// TIA Portal project "Project" (V13)

(* hardware
DEVICE "S7300/ET200M station_1"  S7-300 station
   slot 0: "Rail_0"  Rail  6ES7 390-1***0-0AA0
   slot 1: "PS 307 2A_1"  PS 307 2A  6ES7 307-1BA00-0AA0
   slot 2: "PLC-241"  CPU 315-2 PN/DP  6ES7 315-2EH13-0AB0  V2.6
      slot 1: "MPI/DP interface_1"  X1
      slot 2: "PROFINET interface_1"  PN-IO
         slot 1: "Port_1"  Port
   slot 4: "DI 16/DO 16x24VDC/0.5A_1"  DI16/DO16 x 24V / 0.5A  6ES7 323-1BL00-0AA0
DEVICE "PC-System_1"  SIMATIC PC station
   slot 0: "SIMATIC PC station"  Rail  SIMATIC PC-Station  V1.0
      slot 125: "Stationmanager"  Station_Manager  V6.0.4
   slot 1: "HMI_RT_1"  WinCC RT Advanced  6AV2 104-0xxxx-xxxx  13.0.1.0
      slot 33792: "Host interface"  Host interface
   slot 2: "IE general_1"  IE General  IE_CP  V8.2.0
*)

// ===== PLC "PLC-241"  CPU 315-2 PN/DP =====

VAR_GLOBAL   // PLC tag table "Default tag table"
   "tipka_crna_L_zgoraj" AT %I1.4 : Bool;
   "tipka_crna_L_spodaj" AT %I1.5 : Bool;
   "tipka_crna_D_zgoraj" AT %I1.6 : Bool;
   "tipka_crna_D_spodaj" AT %I1.7 : Bool;
   "kljuc" AT %I1.2 : Bool;
   "tipka_zelena" AT %I1.3 : Bool;
   "vrtljivaMiza_R_vhod" AT %I0.0 : Bool;
   "vrtljivaMiza_I_vhod" AT %I0.1 : Bool;
   "teleskopskaRoka_R_vhod" AT %I0.2 : Bool;
   "teleskopskaRoka_I_vhod" AT %I0.3 : Bool;
   "dvig_R_vhod" AT %I0.4 : Bool;
   "dvig_I_vhod" AT %I0.5 : Bool;
   "prijemalo_R_vhod" AT %I0.6 : Bool;
   "prijemalo_I_vhod" AT %I0.7 : Bool;
   "vrtljivaMiza_S_izhod" AT %Q0.0 : Bool;
   "vrtljivaMiza_P_izhod" AT %Q0.1 : Bool;
   "teleskopskaRoka_S_izhod" AT %Q0.2 : Bool;
   "teleskopskaRoka_P_izhod" AT %Q0.3 : Bool;
   "dvig_S_izhod" AT %Q0.4 : Bool;
   "dvig_P_izhod" AT %Q0.5 : Bool;
   "prijemalo_S_izhod" AT %Q0.6 : Bool;
   "prijemalo_P_izhod" AT %Q0.7 : Bool;
   "lucka_rdeca_L" AT %Q1.4 : Bool;
   "lucka_rumena_L" AT %Q1.5 : Bool;
   "lucka_rdeca_D" AT %Q1.6 : Bool;
   "lucka_rumena_D" AT %Q1.7 : Bool;
   "s" AT %M2.0 : Bool;
   "memory_1" AT %M4.0 : Bool;
   "memory_2" AT %M6.0 : Bool;
END_VAR

TYPE "Lokacija"
   STRUCT
      "ID izdelka" : Int;
      koordinate : "Koordinate";
   END_STRUCT;
END_TYPE

TYPE "Koordinate"
   STRUCT
      miza : Int;
      izteg : Int;
      dvig : Int;
      stisk : Int;
   END_STRUCT;
END_TYPE

DATA_BLOCK "spremenljivke"   // DB1
{ S7_Optimized_Access := 'FALSE' }
VERSION : 0.1
   VAR
      smer : Bool;
      premik : Bool;
      auto_motor1_ccw : Bool;
      auto_motor1_cw : Bool;
      izbiraMotorja : Int;
      levo : Bool;
      desno : Bool;
      vrtljivaMiza_TRENUTNO : Int;
      teleskopskaRoka_TRENUTNO : Int;
      dvig_TRENUTNO : Int;
      premik_TRENUTNO : Int;
      dvig_max : Int;
      vrtljivaMiza_max : Int;
      premik_max : Int;
      teleskopskaRoka_MAX : Int;
      Recept_prej : Int;
      stevecLokacij : Int;
      neki : Int;
      izdelekID : Int;
      izbiraRecepta : Int;
      stevecKosov : Int;
      prva_ref_roka : Bool;
      prva_ref_dvig : Bool;
      prva_ref_stisk : Bool;
      prva_ref_miza : Bool;
      prva_rs_dvig : Bool;
      prva_rs_stisk : Bool;
      prva_rs_roka : Bool;
      prva_rs_miza : Bool;
      miza_ok : Bool;
      stisk_ok : Bool;
      roka_ok : Bool;
      dvig_ok : Bool;
      razlika_dvig : Int;
      razlika_miza : Int;
      razlika_stisk : Int;
      razlika_roka : Int;
   END_VAR
BEGIN
END_DATA_BLOCK

DATA_BLOCK "Motor_DB_1"   // DB2
{ S7_Optimized_Access := 'FALSE' }
VERSION : 0.1
// stored: InstanceOfName Motor
"Motor"
BEGIN
END_DATA_BLOCK

DATA_BLOCK "Lokacije"   // DB3
{ S7_Optimized_Access := 'FALSE' }
VERSION : 0.1
   VAR
      lokacija0 : "Lokacija";
      lokacija1 : "Lokacija";
      lokacija2 : "Lokacija";
      lokacija3 : "Lokacija";
      lokacija4 : "Lokacija";
      lokacija5 : "Lokacija";
      lokacija6 : "Lokacija";
      lokacija7 : "Lokacija";
   END_VAR
BEGIN
END_DATA_BLOCK

DATA_BLOCK "vrtljivaMiza_DB"   // DB4
{ S7_Optimized_Access := 'FALSE' }
VERSION : 0.1
// stored: InstanceOfName vrtljivaMiza
"vrtljivaMiza"
BEGIN
END_DATA_BLOCK

DATA_BLOCK "stevecMotorjev_DB_1"   // DB5
{ S7_Optimized_Access := 'FALSE' }
VERSION : 0.1
// stored: InstanceOfName stevecMotorjev
"stevecMotorjev"
BEGIN
END_DATA_BLOCK

DATA_BLOCK "teleskopskaRoka_DB"   // DB6
{ S7_Optimized_Access := 'FALSE' }
VERSION : 0.1
// stored: InstanceOfName teleskopskaRoka
"teleskopskaRoka"
BEGIN
END_DATA_BLOCK

DATA_BLOCK "dvig_DB"   // DB7
{ S7_Optimized_Access := 'FALSE' }
VERSION : 0.1
// stored: InstanceOfName dvig
"dvig"
BEGIN
END_DATA_BLOCK

DATA_BLOCK "prijemalo_DB"   // DB8
{ S7_Optimized_Access := 'FALSE' }
VERSION : 0.1
// stored: InstanceOfName prijemalo
"prijemalo"
BEGIN
END_DATA_BLOCK

DATA_BLOCK "TrenutnaLokacija"   // DB9
{ S7_Optimized_Access := 'FALSE' }
VERSION : 0.1
   VAR
      lokacija : "Lokacija";
   END_VAR
BEGIN
END_DATA_BLOCK

DATA_BLOCK "IzbiraLokacije_DB"   // DB10
{ S7_Optimized_Access := 'FALSE' }
VERSION : 0.1
// stored: InstanceOfName IzbiraLokacije
"IzbiraLokacije"
BEGIN
END_DATA_BLOCK

DATA_BLOCK "IzbiraLokacije_DB_1"   // DB11
{ S7_Optimized_Access := 'FALSE' }
VERSION : 0.1
// stored: InstanceOfName IzbiraLokacije
"IzbiraLokacije"
BEGIN
END_DATA_BLOCK

DATA_BLOCK "Recept 1"   // DB12
{ S7_Optimized_Access := 'FALSE' }
VERSION : 0.1
   VAR
      lokacija10 : "Lokacija";
      lokacija11 : "Lokacija";
      lokacija12 : "Lokacija";
      lokacija13 : "Lokacija";
      lokacija14 : "Lokacija";
      lokacija15 : "Lokacija";
      lokacija16 : "Lokacija";
      lokacija17 : "Lokacija";
   END_VAR
BEGIN
END_DATA_BLOCK

DATA_BLOCK "Recept 2"   // DB13
{ S7_Optimized_Access := 'FALSE' }
VERSION : 0.1
   VAR
      lokacija20 : "Lokacija";
      lokacija21 : "Lokacija";
      lokacija22 : "Lokacija";
      lokacija23 : "Lokacija";
      lokacija24 : "Lokacija";
      lokacija25 : "Lokacija";
      lokacija26 : "Lokacija";
      lokacija27 : "Lokacija";
   END_VAR
BEGIN
END_DATA_BLOCK

DATA_BLOCK "Alarmi"   // DB14
{ S7_Optimized_Access := 'FALSE' }
VERSION : 0.1
   VAR
      alarmi : Array[0..15] of Bool;
      alarmPotrdi : Bool;
      alarmRS1 : Bool;
      alarmRS2 : Bool;
      alarmRS3 : Bool;
      alarmRS4 : Bool;
      alarmRS5 : Bool;
      alarmRS6 : Bool;
      Globalni_alarm : Bool;
   END_VAR
BEGIN
END_DATA_BLOCK

DATA_BLOCK "izbiraAlarmov_DB"   // DB15
{ S7_Optimized_Access := 'FALSE' }
VERSION : 0.1
// stored: InstanceOfName izbiraAlarmov
"izbiraAlarmov"
BEGIN
END_DATA_BLOCK

FUNCTION_BLOCK "Motor"   // FB1, LAD
{ S7_Optimized_Access := 'FALSE' }
VERSION : 0.1
   VAR_TEMP   // added for the SCL form of the ladder/FBD networks
      _w1 : Bool;
      _w2 : Bool;
   END_VAR
BEGIN

REGION Network 1
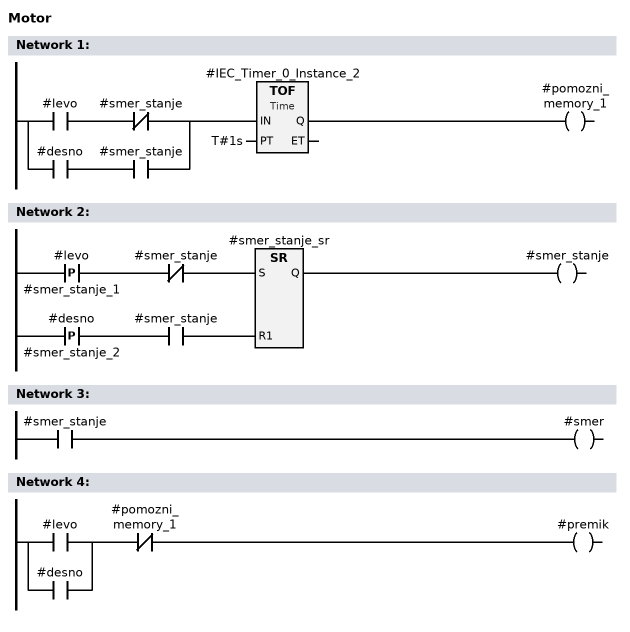
   #IEC_Timer_0_Instance_2.TOF(IN := (#levo AND NOT #smer_stanje) OR (#desno AND #smer_stanje), PT := T#1s);
   #pomozni_memory_1 := #IEC_Timer_0_Instance_2.Q;
END_REGION

REGION Network 2
   RUNG wire#powerrail
      P_Contact(operand := #levo, bit := #smer_stanje_1)
      I_Contact( #smer_stanje )
      S_SR(operand := #smer_stanje_sr, r1 := wire#w1)
      Coil( #smer_stanje )
   END_RUNG
   RUNG wire#powerrail
      P_Contact(operand := #desno, bit := #smer_stanje_2)
      Contact( #smer_stanje )
   END_RUNG wire#w1
   // the same network as SCL:
   #_w1 := #levo AND NOT #smer_stanje_1;   // rising edge of #levo
   #smer_stanje_1 := #levo;
   #_w2 := #desno AND NOT #smer_stanje_2;   // rising edge of #desno
   #smer_stanje_2 := #desno;
   IF #_w1 AND NOT #smer_stanje THEN
       #smer_stanje_sr := TRUE;   // SR flip-flop
   END_IF;
   IF #_w2 AND #smer_stanje THEN #smer_stanje_sr := FALSE; END_IF;
   #smer_stanje := #smer_stanje_sr;
END_REGION

REGION Network 3
   RUNG wire#powerrail
      Contact( #smer_stanje )
      Coil( #smer )
   END_RUNG
   // the same network as SCL:
   #smer := #smer_stanje;
END_REGION

REGION Network 4
   RUNG wire#powerrail
      Contact( #levo )
      wire#w1
      I_Contact( #pomozni_memory_1 )
      Coil( #premik )
   END_RUNG
   RUNG wire#powerrail
      Contact( #desno )
   END_RUNG wire#w1
   // the same network as SCL:
   #premik := (#levo OR #desno) AND NOT #pomozni_memory_1;
END_REGION
END_FUNCTION_BLOCK

FUNCTION_BLOCK "stevecMotorjev"   // FB2, LAD
{ S7_Optimized_Access := 'FALSE' }
VERSION : 0.1
BEGIN

REGION Network 1
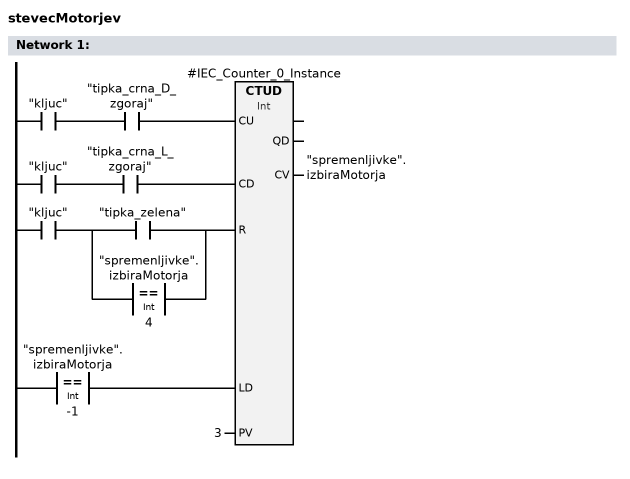
   #IEC_Counter_0_Instance.CTUD(CU := "kljuc" AND "tipka_crna_D_zgoraj",
                           CD := "kljuc" AND "tipka_crna_L_zgoraj",
                           R := "kljuc" AND ("tipka_zelena" OR ("spremenljivke".izbiraMotorja = 4)),
                           LD := "spremenljivke".izbiraMotorja = (-1),
                           PV := 3,
                           CV => "spremenljivke".izbiraMotorja);
END_REGION
END_FUNCTION_BLOCK

FUNCTION_BLOCK "vrtljivaMiza"   // FB3, LAD
{ S7_Optimized_Access := 'FALSE' }
VERSION : 0.1
BEGIN

REGION Network 1
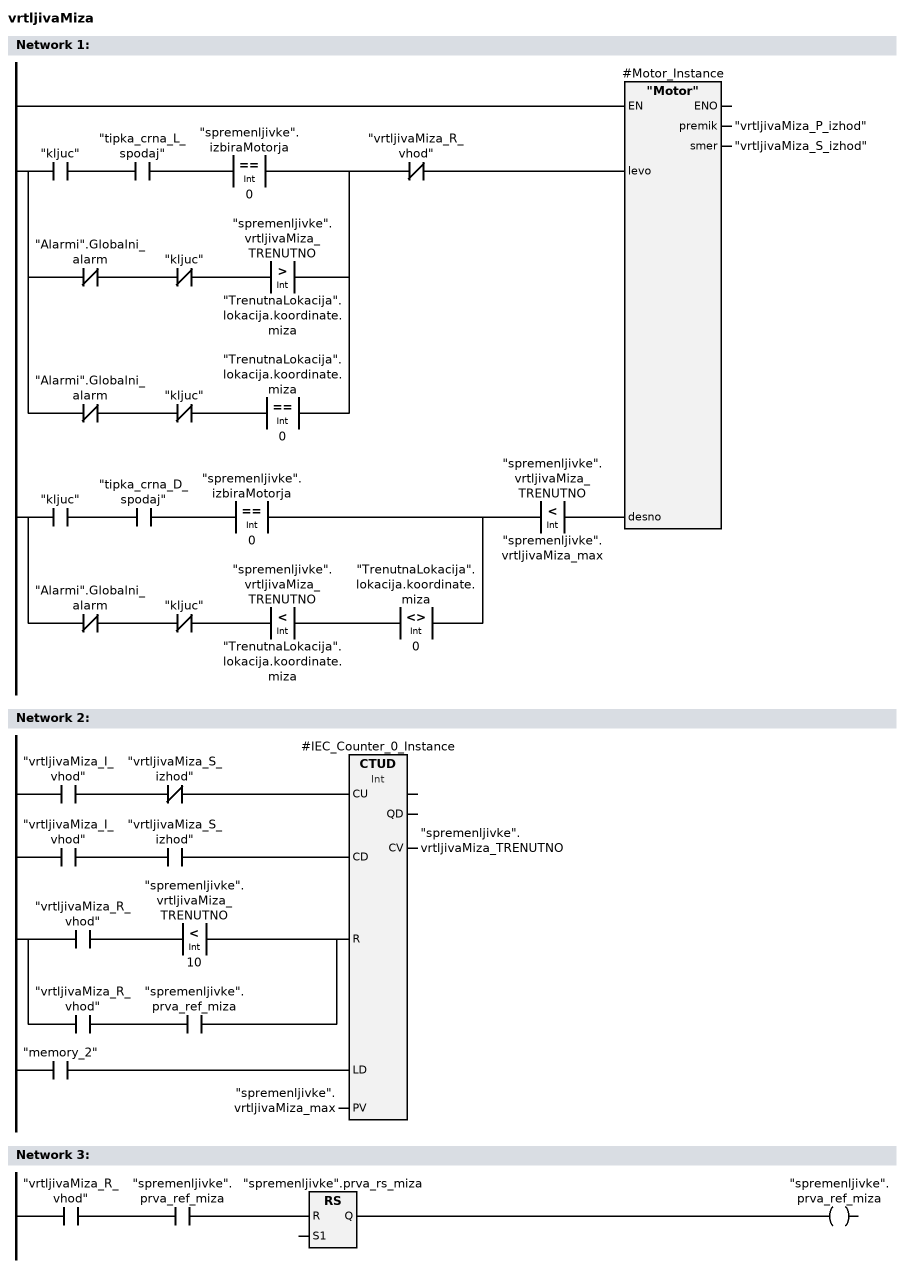
   RUNG wire#powerrail
      #Motor_Instance(levo := wire#w2, desno := wire#w4, premik => "vrtljivaMiza_P_izhod", smer => "vrtljivaMiza_S_izhod")
   END_RUNG
   RUNG wire#powerrail
      Contact( "kljuc" )
      Contact( "tipka_crna_L_spodaj" )
      { S7_Templates := "SrcType := Int" } EQ_Contact(in1 := "spremenljivke".izbiraMotorja, in2 := 0)
      wire#w1
      I_Contact( "vrtljivaMiza_R_vhod" )
   END_RUNG wire#w2
   RUNG wire#powerrail
      I_Contact( "Alarmi".Globalni_alarm )
      I_Contact( "kljuc" )
      { S7_Templates := "SrcType := Int" } GT_Contact(in1 := "spremenljivke".vrtljivaMiza_TRENUTNO, in2 := "TrenutnaLokacija".lokacija.koordinate.miza)
   END_RUNG wire#w1
   RUNG wire#powerrail
      I_Contact( "Alarmi".Globalni_alarm )
      I_Contact( "kljuc" )
      { S7_Templates := "SrcType := Int" } EQ_Contact(in1 := "TrenutnaLokacija".lokacija.koordinate.miza, in2 := 0)
   END_RUNG wire#w1
   RUNG wire#powerrail
      Contact( "kljuc" )
      Contact( "tipka_crna_D_spodaj" )
      { S7_Templates := "SrcType := Int" } EQ_Contact(in1 := "spremenljivke".izbiraMotorja, in2 := 0)
      wire#w3
      { S7_Templates := "SrcType := Int" } LT_Contact(in1 := "spremenljivke".vrtljivaMiza_TRENUTNO, in2 := "spremenljivke".vrtljivaMiza_max)
   END_RUNG wire#w4
   RUNG wire#powerrail
      I_Contact( "Alarmi".Globalni_alarm )
      I_Contact( "kljuc" )
      { S7_Templates := "SrcType := Int" } LT_Contact(in1 := "spremenljivke".vrtljivaMiza_TRENUTNO, in2 := "TrenutnaLokacija".lokacija.koordinate.miza)
      { S7_Templates := "SrcType := Int" } NE_Contact(in1 := "TrenutnaLokacija".lokacija.koordinate.miza, in2 := 0)
   END_RUNG wire#w3
   // the same network as SCL:
   #Motor_Instance(levo := (("kljuc" AND "tipka_crna_L_spodaj" AND ("spremenljivke".izbiraMotorja = 0)) OR (NOT "Alarmi".Globalni_alarm AND NOT "kljuc" AND ("spremenljivke".vrtljivaMiza_TRENUTNO > "TrenutnaLokacija".lokacija.koordinate.miza)) OR (NOT "Alarmi".Globalni_alarm AND NOT "kljuc" AND ("TrenutnaLokacija".lokacija.koordinate.miza = 0))) AND NOT "vrtljivaMiza_R_vhod",   // "Motor"
                   desno := (("kljuc" AND "tipka_crna_D_spodaj" AND ("spremenljivke".izbiraMotorja = 0)) OR (NOT "Alarmi".Globalni_alarm AND NOT "kljuc" AND ("spremenljivke".vrtljivaMiza_TRENUTNO < "TrenutnaLokacija".lokacija.koordinate.miza) AND ("TrenutnaLokacija".lokacija.koordinate.miza <> 0))) AND ("spremenljivke".vrtljivaMiza_TRENUTNO < "spremenljivke".vrtljivaMiza_max),
                   premik => "vrtljivaMiza_P_izhod",
                   smer => "vrtljivaMiza_S_izhod");
END_REGION

REGION Network 2
   #IEC_Counter_0_Instance.CTUD(CU := "vrtljivaMiza_I_vhod" AND NOT "vrtljivaMiza_S_izhod",
                           CD := "vrtljivaMiza_I_vhod" AND "vrtljivaMiza_S_izhod",
                           R := ("vrtljivaMiza_R_vhod" AND ("spremenljivke".vrtljivaMiza_TRENUTNO < 10)) OR ("vrtljivaMiza_R_vhod" AND "spremenljivke".prva_ref_miza),
                           LD := "memory_2",
                           PV := "spremenljivke".vrtljivaMiza_max,
                           CV => "spremenljivke".vrtljivaMiza_TRENUTNO);
END_REGION

REGION Network 3
   RUNG wire#powerrail
      Contact( "vrtljivaMiza_R_vhod" )
      Contact( "spremenljivke".prva_ref_miza )
      S_RS(operand := "spremenljivke".prva_rs_miza, s1 :=)
      Coil( "spremenljivke".prva_ref_miza )
   END_RUNG
   // the same network as SCL:
   IF "vrtljivaMiza_R_vhod" AND "spremenljivke".prva_ref_miza THEN
       "spremenljivke".prva_rs_miza := FALSE;   // RS flip-flop
   END_IF;
   "spremenljivke".prva_ref_miza := "spremenljivke".prva_rs_miza;
END_REGION
END_FUNCTION_BLOCK

FUNCTION_BLOCK "teleskopskaRoka"   // FB4, LAD
{ S7_Optimized_Access := 'FALSE' }
VERSION : 0.1
BEGIN

REGION Network 1
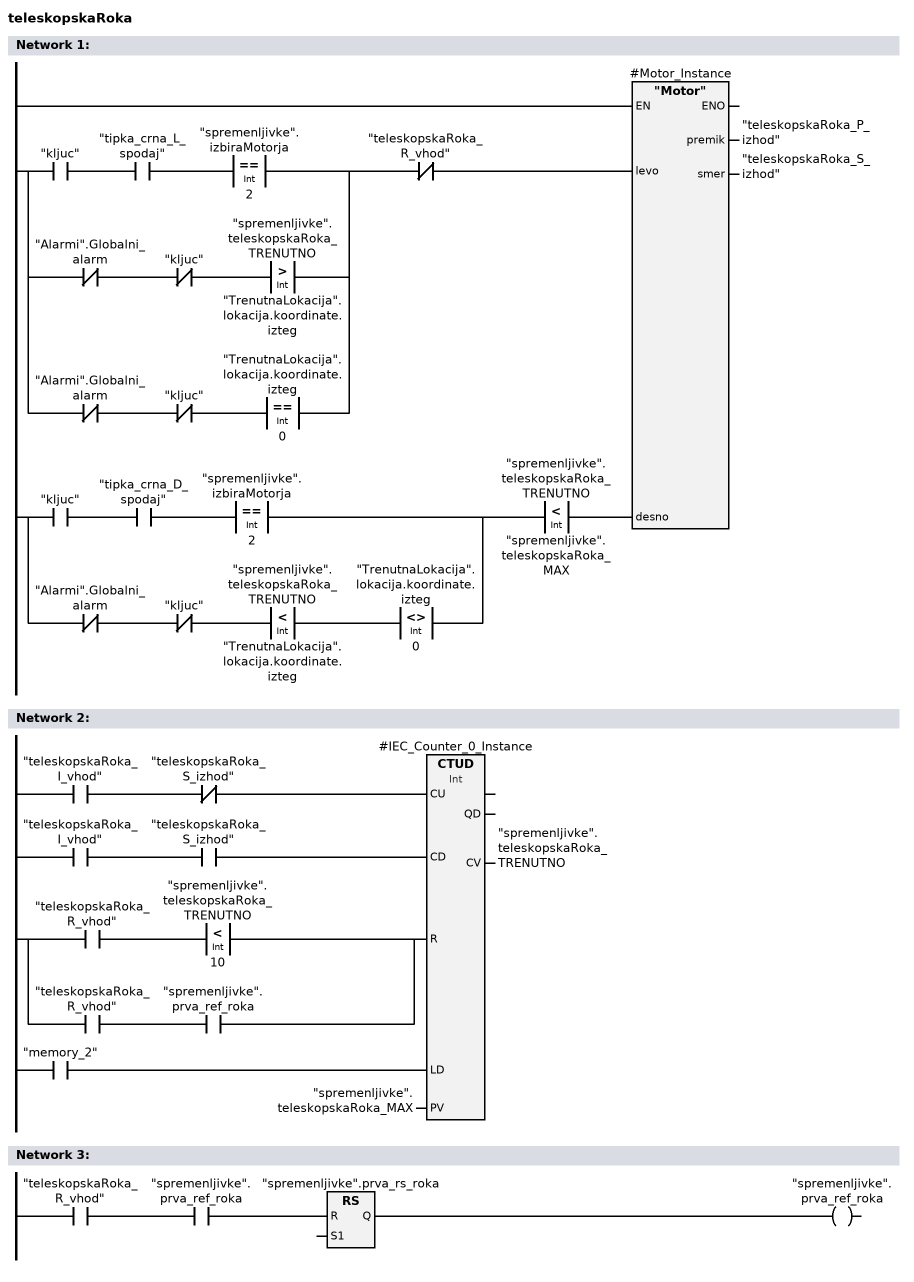
   RUNG wire#powerrail
      #Motor_Instance(levo := wire#w2, desno := wire#w4, premik => "teleskopskaRoka_P_izhod", smer => "teleskopskaRoka_S_izhod")
   END_RUNG
   RUNG wire#powerrail
      Contact( "kljuc" )
      Contact( "tipka_crna_L_spodaj" )
      { S7_Templates := "SrcType := Int" } EQ_Contact(in1 := "spremenljivke".izbiraMotorja, in2 := 2)
      wire#w1
      I_Contact( "teleskopskaRoka_R_vhod" )
   END_RUNG wire#w2
   RUNG wire#powerrail
      I_Contact( "Alarmi".Globalni_alarm )
      I_Contact( "kljuc" )
      { S7_Templates := "SrcType := Int" } GT_Contact(in1 := "spremenljivke".teleskopskaRoka_TRENUTNO, in2 := "TrenutnaLokacija".lokacija.koordinate.izteg)
   END_RUNG wire#w1
   RUNG wire#powerrail
      I_Contact( "Alarmi".Globalni_alarm )
      I_Contact( "kljuc" )
      { S7_Templates := "SrcType := Int" } EQ_Contact(in1 := "TrenutnaLokacija".lokacija.koordinate.izteg, in2 := 0)
   END_RUNG wire#w1
   RUNG wire#powerrail
      Contact( "kljuc" )
      Contact( "tipka_crna_D_spodaj" )
      { S7_Templates := "SrcType := Int" } EQ_Contact(in1 := "spremenljivke".izbiraMotorja, in2 := 2)
      wire#w3
      { S7_Templates := "SrcType := Int" } LT_Contact(in1 := "spremenljivke".teleskopskaRoka_TRENUTNO, in2 := "spremenljivke".teleskopskaRoka_MAX)
   END_RUNG wire#w4
   RUNG wire#powerrail
      I_Contact( "Alarmi".Globalni_alarm )
      I_Contact( "kljuc" )
      { S7_Templates := "SrcType := Int" } LT_Contact(in1 := "spremenljivke".teleskopskaRoka_TRENUTNO, in2 := "TrenutnaLokacija".lokacija.koordinate.izteg)
      { S7_Templates := "SrcType := Int" } NE_Contact(in1 := "TrenutnaLokacija".lokacija.koordinate.izteg, in2 := 0)
   END_RUNG wire#w3
   // the same network as SCL:
   #Motor_Instance(levo := (("kljuc" AND "tipka_crna_L_spodaj" AND ("spremenljivke".izbiraMotorja = 2)) OR (NOT "Alarmi".Globalni_alarm AND NOT "kljuc" AND ("spremenljivke".teleskopskaRoka_TRENUTNO > "TrenutnaLokacija".lokacija.koordinate.izteg)) OR (NOT "Alarmi".Globalni_alarm AND NOT "kljuc" AND ("TrenutnaLokacija".lokacija.koordinate.izteg = 0))) AND NOT "teleskopskaRoka_R_vhod",   // "Motor"
                   desno := (("kljuc" AND "tipka_crna_D_spodaj" AND ("spremenljivke".izbiraMotorja = 2)) OR (NOT "Alarmi".Globalni_alarm AND NOT "kljuc" AND ("spremenljivke".teleskopskaRoka_TRENUTNO < "TrenutnaLokacija".lokacija.koordinate.izteg) AND ("TrenutnaLokacija".lokacija.koordinate.izteg <> 0))) AND ("spremenljivke".teleskopskaRoka_TRENUTNO < "spremenljivke".teleskopskaRoka_MAX),
                   premik => "teleskopskaRoka_P_izhod",
                   smer => "teleskopskaRoka_S_izhod");
END_REGION

REGION Network 2
   #IEC_Counter_0_Instance.CTUD(CU := "teleskopskaRoka_I_vhod" AND NOT "teleskopskaRoka_S_izhod",
                           CD := "teleskopskaRoka_I_vhod" AND "teleskopskaRoka_S_izhod",
                           R := ("teleskopskaRoka_R_vhod" AND ("spremenljivke".teleskopskaRoka_TRENUTNO < 10)) OR ("teleskopskaRoka_R_vhod" AND "spremenljivke".prva_ref_roka),
                           LD := "memory_2",
                           PV := "spremenljivke".teleskopskaRoka_MAX,
                           CV => "spremenljivke".teleskopskaRoka_TRENUTNO);
END_REGION

REGION Network 3
   RUNG wire#powerrail
      Contact( "teleskopskaRoka_R_vhod" )
      Contact( "spremenljivke".prva_ref_roka )
      S_RS(operand := "spremenljivke".prva_rs_roka, s1 :=)
      Coil( "spremenljivke".prva_ref_roka )
   END_RUNG
   // the same network as SCL:
   IF "teleskopskaRoka_R_vhod" AND "spremenljivke".prva_ref_roka THEN
       "spremenljivke".prva_rs_roka := FALSE;   // RS flip-flop
   END_IF;
   "spremenljivke".prva_ref_roka := "spremenljivke".prva_rs_roka;
END_REGION
END_FUNCTION_BLOCK

FUNCTION_BLOCK "dvig"   // FB5, LAD
{ S7_Optimized_Access := 'FALSE' }
VERSION : 0.1
BEGIN

REGION Network 1
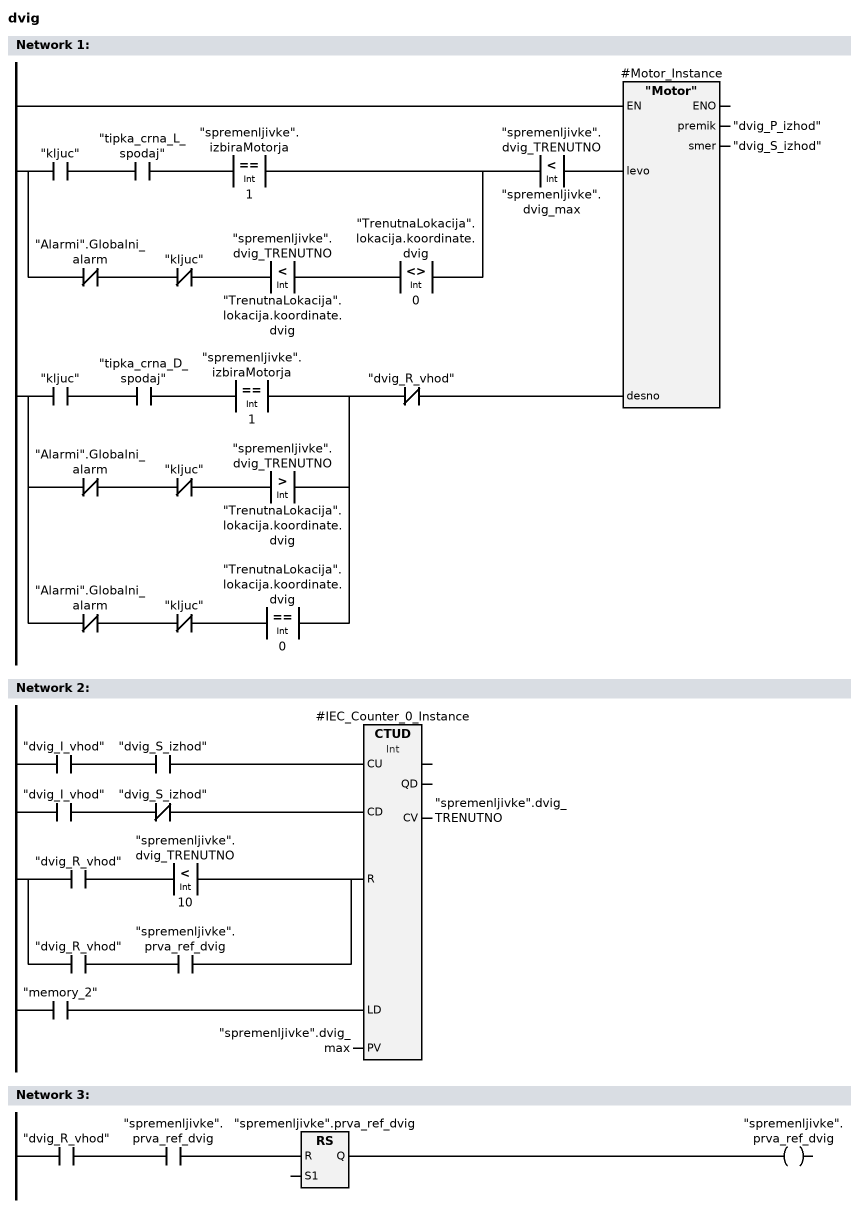
   RUNG wire#powerrail
      #Motor_Instance(levo := wire#w2, desno := wire#w4, premik => "dvig_P_izhod", smer => "dvig_S_izhod")
   END_RUNG
   RUNG wire#powerrail
      Contact( "kljuc" )
      Contact( "tipka_crna_L_spodaj" )
      { S7_Templates := "SrcType := Int" } EQ_Contact(in1 := "spremenljivke".izbiraMotorja, in2 := 1)
      wire#w1
      { S7_Templates := "SrcType := Int" } LT_Contact(in1 := "spremenljivke".dvig_TRENUTNO, in2 := "spremenljivke".dvig_max)
   END_RUNG wire#w2
   RUNG wire#powerrail
      I_Contact( "Alarmi".Globalni_alarm )
      I_Contact( "kljuc" )
      { S7_Templates := "SrcType := Int" } LT_Contact(in1 := "spremenljivke".dvig_TRENUTNO, in2 := "TrenutnaLokacija".lokacija.koordinate.dvig)
      { S7_Templates := "SrcType := Int" } NE_Contact(in1 := "TrenutnaLokacija".lokacija.koordinate.dvig, in2 := 0)
   END_RUNG wire#w1
   RUNG wire#powerrail
      Contact( "kljuc" )
      Contact( "tipka_crna_D_spodaj" )
      { S7_Templates := "SrcType := Int" } EQ_Contact(in1 := "spremenljivke".izbiraMotorja, in2 := 1)
      wire#w3
      I_Contact( "dvig_R_vhod" )
   END_RUNG wire#w4
   RUNG wire#powerrail
      I_Contact( "Alarmi".Globalni_alarm )
      I_Contact( "kljuc" )
      { S7_Templates := "SrcType := Int" } GT_Contact(in1 := "spremenljivke".dvig_TRENUTNO, in2 := "TrenutnaLokacija".lokacija.koordinate.dvig)
   END_RUNG wire#w3
   RUNG wire#powerrail
      I_Contact( "Alarmi".Globalni_alarm )
      I_Contact( "kljuc" )
      { S7_Templates := "SrcType := Int" } EQ_Contact(in1 := "TrenutnaLokacija".lokacija.koordinate.dvig, in2 := 0)
   END_RUNG wire#w3
   // the same network as SCL:
   #Motor_Instance(levo := (("kljuc" AND "tipka_crna_L_spodaj" AND ("spremenljivke".izbiraMotorja = 1)) OR (NOT "Alarmi".Globalni_alarm AND NOT "kljuc" AND ("spremenljivke".dvig_TRENUTNO < "TrenutnaLokacija".lokacija.koordinate.dvig) AND ("TrenutnaLokacija".lokacija.koordinate.dvig <> 0))) AND ("spremenljivke".dvig_TRENUTNO < "spremenljivke".dvig_max),   // "Motor"
                   desno := (("kljuc" AND "tipka_crna_D_spodaj" AND ("spremenljivke".izbiraMotorja = 1)) OR (NOT "Alarmi".Globalni_alarm AND NOT "kljuc" AND ("spremenljivke".dvig_TRENUTNO > "TrenutnaLokacija".lokacija.koordinate.dvig)) OR (NOT "Alarmi".Globalni_alarm AND NOT "kljuc" AND ("TrenutnaLokacija".lokacija.koordinate.dvig = 0))) AND NOT "dvig_R_vhod",
                   premik => "dvig_P_izhod",
                   smer => "dvig_S_izhod");
END_REGION

REGION Network 2
   #IEC_Counter_0_Instance.CTUD(CU := "dvig_I_vhod" AND "dvig_S_izhod",
                           CD := "dvig_I_vhod" AND NOT "dvig_S_izhod",
                           R := ("dvig_R_vhod" AND ("spremenljivke".dvig_TRENUTNO < 10)) OR ("dvig_R_vhod" AND "spremenljivke".prva_ref_dvig),
                           LD := "memory_2",
                           PV := "spremenljivke".dvig_max,
                           CV => "spremenljivke".dvig_TRENUTNO);
END_REGION

REGION Network 3
   RUNG wire#powerrail
      Contact( "dvig_R_vhod" )
      Contact( "spremenljivke".prva_ref_dvig )
      S_RS(operand := "spremenljivke".prva_ref_dvig, s1 :=)
      Coil( "spremenljivke".prva_ref_dvig )
   END_RUNG
   // the same network as SCL:
   IF "dvig_R_vhod" AND "spremenljivke".prva_ref_dvig THEN
       "spremenljivke".prva_ref_dvig := FALSE;   // RS flip-flop
   END_IF;
   "spremenljivke".prva_ref_dvig := "spremenljivke".prva_ref_dvig;
END_REGION
END_FUNCTION_BLOCK

FUNCTION_BLOCK "prijemalo"   // FB6, LAD
{ S7_Optimized_Access := 'FALSE' }
VERSION : 0.1
BEGIN

REGION Network 1
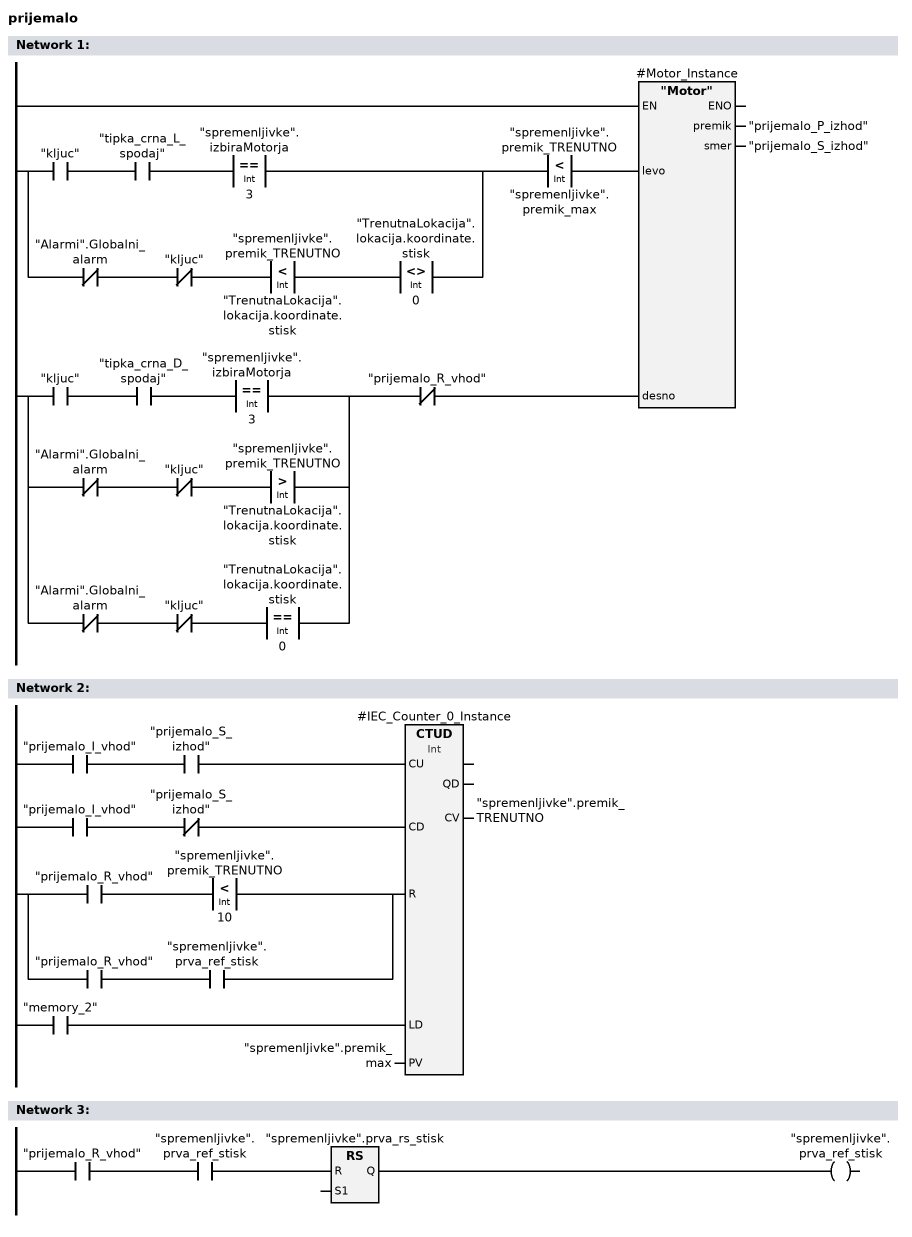
   RUNG wire#powerrail
      #Motor_Instance(levo := wire#w2, desno := wire#w4, premik => "prijemalo_P_izhod", smer => "prijemalo_S_izhod")
   END_RUNG
   RUNG wire#powerrail
      Contact( "kljuc" )
      Contact( "tipka_crna_L_spodaj" )
      { S7_Templates := "SrcType := Int" } EQ_Contact(in1 := "spremenljivke".izbiraMotorja, in2 := 3)
      wire#w1
      { S7_Templates := "SrcType := Int" } LT_Contact(in1 := "spremenljivke".premik_TRENUTNO, in2 := "spremenljivke".premik_max)
   END_RUNG wire#w2
   RUNG wire#powerrail
      I_Contact( "Alarmi".Globalni_alarm )
      I_Contact( "kljuc" )
      { S7_Templates := "SrcType := Int" } LT_Contact(in1 := "spremenljivke".premik_TRENUTNO, in2 := "TrenutnaLokacija".lokacija.koordinate.stisk)
      { S7_Templates := "SrcType := Int" } NE_Contact(in1 := "TrenutnaLokacija".lokacija.koordinate.stisk, in2 := 0)
   END_RUNG wire#w1
   RUNG wire#powerrail
      Contact( "kljuc" )
      Contact( "tipka_crna_D_spodaj" )
      { S7_Templates := "SrcType := Int" } EQ_Contact(in1 := "spremenljivke".izbiraMotorja, in2 := 3)
      wire#w3
      I_Contact( "prijemalo_R_vhod" )
   END_RUNG wire#w4
   RUNG wire#powerrail
      I_Contact( "Alarmi".Globalni_alarm )
      I_Contact( "kljuc" )
      { S7_Templates := "SrcType := Int" } GT_Contact(in1 := "spremenljivke".premik_TRENUTNO, in2 := "TrenutnaLokacija".lokacija.koordinate.stisk)
   END_RUNG wire#w3
   RUNG wire#powerrail
      I_Contact( "Alarmi".Globalni_alarm )
      I_Contact( "kljuc" )
      { S7_Templates := "SrcType := Int" } EQ_Contact(in1 := "TrenutnaLokacija".lokacija.koordinate.stisk, in2 := 0)
   END_RUNG wire#w3
   // the same network as SCL:
   #Motor_Instance(levo := (("kljuc" AND "tipka_crna_L_spodaj" AND ("spremenljivke".izbiraMotorja = 3)) OR (NOT "Alarmi".Globalni_alarm AND NOT "kljuc" AND ("spremenljivke".premik_TRENUTNO < "TrenutnaLokacija".lokacija.koordinate.stisk) AND ("TrenutnaLokacija".lokacija.koordinate.stisk <> 0))) AND ("spremenljivke".premik_TRENUTNO < "spremenljivke".premik_max),   // "Motor"
                   desno := (("kljuc" AND "tipka_crna_D_spodaj" AND ("spremenljivke".izbiraMotorja = 3)) OR (NOT "Alarmi".Globalni_alarm AND NOT "kljuc" AND ("spremenljivke".premik_TRENUTNO > "TrenutnaLokacija".lokacija.koordinate.stisk)) OR (NOT "Alarmi".Globalni_alarm AND NOT "kljuc" AND ("TrenutnaLokacija".lokacija.koordinate.stisk = 0))) AND NOT "prijemalo_R_vhod",
                   premik => "prijemalo_P_izhod",
                   smer => "prijemalo_S_izhod");
END_REGION

REGION Network 2
   #IEC_Counter_0_Instance.CTUD(CU := "prijemalo_I_vhod" AND "prijemalo_S_izhod",
                           CD := "prijemalo_I_vhod" AND NOT "prijemalo_S_izhod",
                           R := ("prijemalo_R_vhod" AND ("spremenljivke".premik_TRENUTNO < 10)) OR ("prijemalo_R_vhod" AND "spremenljivke".prva_ref_stisk),
                           LD := "memory_2",
                           PV := "spremenljivke".premik_max,
                           CV => "spremenljivke".premik_TRENUTNO);
END_REGION

REGION Network 3
   RUNG wire#powerrail
      Contact( "prijemalo_R_vhod" )
      Contact( "spremenljivke".prva_ref_stisk )
      S_RS(operand := "spremenljivke".prva_rs_stisk, s1 :=)
      Coil( "spremenljivke".prva_ref_stisk )
   END_RUNG
   // the same network as SCL:
   IF "prijemalo_R_vhod" AND "spremenljivke".prva_ref_stisk THEN
       "spremenljivke".prva_rs_stisk := FALSE;   // RS flip-flop
   END_IF;
   "spremenljivke".prva_ref_stisk := "spremenljivke".prva_rs_stisk;
END_REGION
END_FUNCTION_BLOCK

FUNCTION_BLOCK "IzbiraLokacije"   // FB7, LAD
{ S7_Optimized_Access := 'FALSE' }
VERSION : 0.1
   VAR_TEMP   // added for the SCL form of the ladder/FBD networks
      _w1 : Bool;
   END_VAR
BEGIN

REGION Network 1
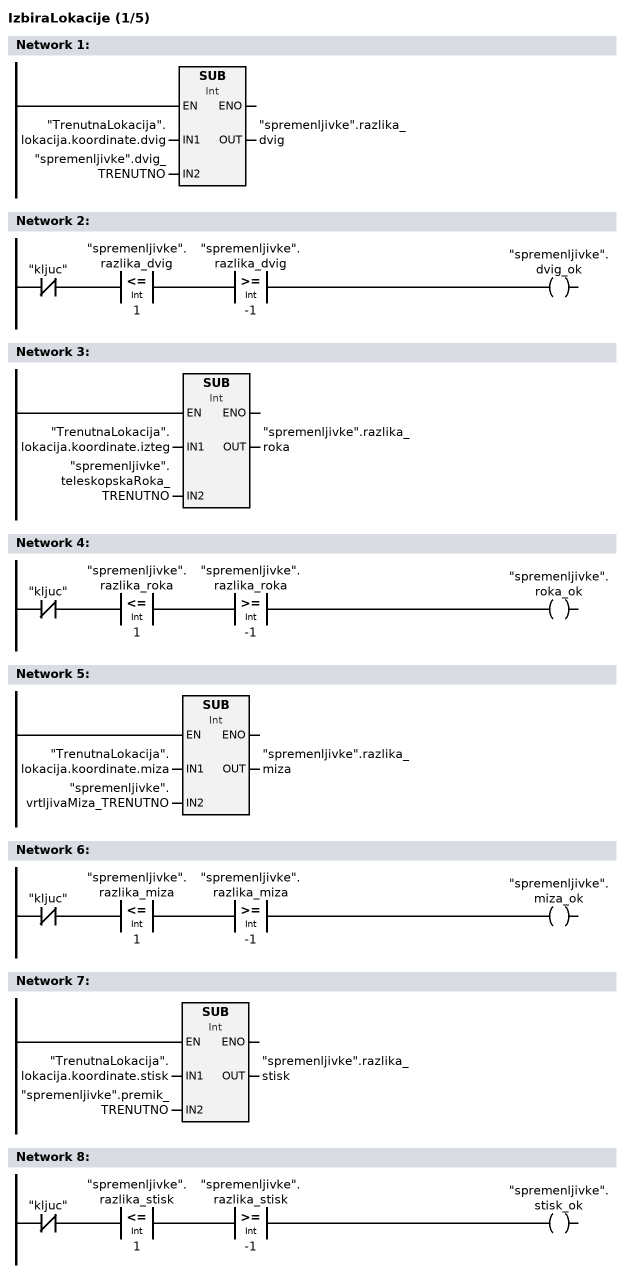
   RUNG wire#powerrail
      { S7_Templates := "SrcType := Int"; S7_GenerateENO := "TRUE" } Sub(in1 := "TrenutnaLokacija".lokacija.koordinate.dvig, in2 := "spremenljivke".dvig_TRENUTNO, out => "spremenljivke".razlika_dvig)
   END_RUNG
   // the same network as SCL:
   "spremenljivke".razlika_dvig := "TrenutnaLokacija".lokacija.koordinate.dvig - "spremenljivke".dvig_TRENUTNO;
END_REGION

REGION Network 2
   RUNG wire#powerrail
      I_Contact( "kljuc" )
      { S7_Templates := "SrcType := Int" } LE_Contact(in1 := "spremenljivke".razlika_dvig, in2 := 1)
      { S7_Templates := "SrcType := Int" } GE_Contact(in1 := "spremenljivke".razlika_dvig, in2 := -1)
      Coil( "spremenljivke".dvig_ok )
   END_RUNG
   // the same network as SCL:
   "spremenljivke".dvig_ok := NOT "kljuc" AND ("spremenljivke".razlika_dvig <= 1) AND ("spremenljivke".razlika_dvig >= (-1));
END_REGION

REGION Network 3
   RUNG wire#powerrail
      { S7_Templates := "SrcType := Int"; S7_GenerateENO := "TRUE" } Sub(in1 := "TrenutnaLokacija".lokacija.koordinate.izteg, in2 := "spremenljivke".teleskopskaRoka_TRENUTNO, out => "spremenljivke".razlika_roka)
   END_RUNG
   // the same network as SCL:
   "spremenljivke".razlika_roka := "TrenutnaLokacija".lokacija.koordinate.izteg - "spremenljivke".teleskopskaRoka_TRENUTNO;
END_REGION

REGION Network 4
   RUNG wire#powerrail
      I_Contact( "kljuc" )
      { S7_Templates := "SrcType := Int" } LE_Contact(in1 := "spremenljivke".razlika_roka, in2 := 1)
      { S7_Templates := "SrcType := Int" } GE_Contact(in1 := "spremenljivke".razlika_roka, in2 := -1)
      Coil( "spremenljivke".roka_ok )
   END_RUNG
   // the same network as SCL:
   "spremenljivke".roka_ok := NOT "kljuc" AND ("spremenljivke".razlika_roka <= 1) AND ("spremenljivke".razlika_roka >= (-1));
END_REGION

REGION Network 5
   RUNG wire#powerrail
      { S7_Templates := "SrcType := Int"; S7_GenerateENO := "TRUE" } Sub(in1 := "TrenutnaLokacija".lokacija.koordinate.miza, in2 := "spremenljivke".vrtljivaMiza_TRENUTNO, out => "spremenljivke".razlika_miza)
   END_RUNG
   // the same network as SCL:
   "spremenljivke".razlika_miza := "TrenutnaLokacija".lokacija.koordinate.miza - "spremenljivke".vrtljivaMiza_TRENUTNO;
END_REGION

REGION Network 6
   RUNG wire#powerrail
      I_Contact( "kljuc" )
      { S7_Templates := "SrcType := Int" } LE_Contact(in1 := "spremenljivke".razlika_miza, in2 := 1)
      { S7_Templates := "SrcType := Int" } GE_Contact(in1 := "spremenljivke".razlika_miza, in2 := -1)
      Coil( "spremenljivke".miza_ok )
   END_RUNG
   // the same network as SCL:
   "spremenljivke".miza_ok := NOT "kljuc" AND ("spremenljivke".razlika_miza <= 1) AND ("spremenljivke".razlika_miza >= (-1));
END_REGION

REGION Network 7
   RUNG wire#powerrail
      { S7_Templates := "SrcType := Int"; S7_GenerateENO := "TRUE" } Sub(in1 := "TrenutnaLokacija".lokacija.koordinate.stisk, in2 := "spremenljivke".premik_TRENUTNO, out => "spremenljivke".razlika_stisk)
   END_RUNG
   // the same network as SCL:
   "spremenljivke".razlika_stisk := "TrenutnaLokacija".lokacija.koordinate.stisk - "spremenljivke".premik_TRENUTNO;
END_REGION

REGION Network 8
   RUNG wire#powerrail
      I_Contact( "kljuc" )
      { S7_Templates := "SrcType := Int" } LE_Contact(in1 := "spremenljivke".razlika_stisk, in2 := 1)
      { S7_Templates := "SrcType := Int" } GE_Contact(in1 := "spremenljivke".razlika_stisk, in2 := -1)
      Coil( "spremenljivke".stisk_ok )
   END_RUNG
   // the same network as SCL:
   "spremenljivke".stisk_ok := NOT "kljuc" AND ("spremenljivke".razlika_stisk <= 1) AND ("spremenljivke".razlika_stisk >= (-1));
END_REGION

REGION Network 9
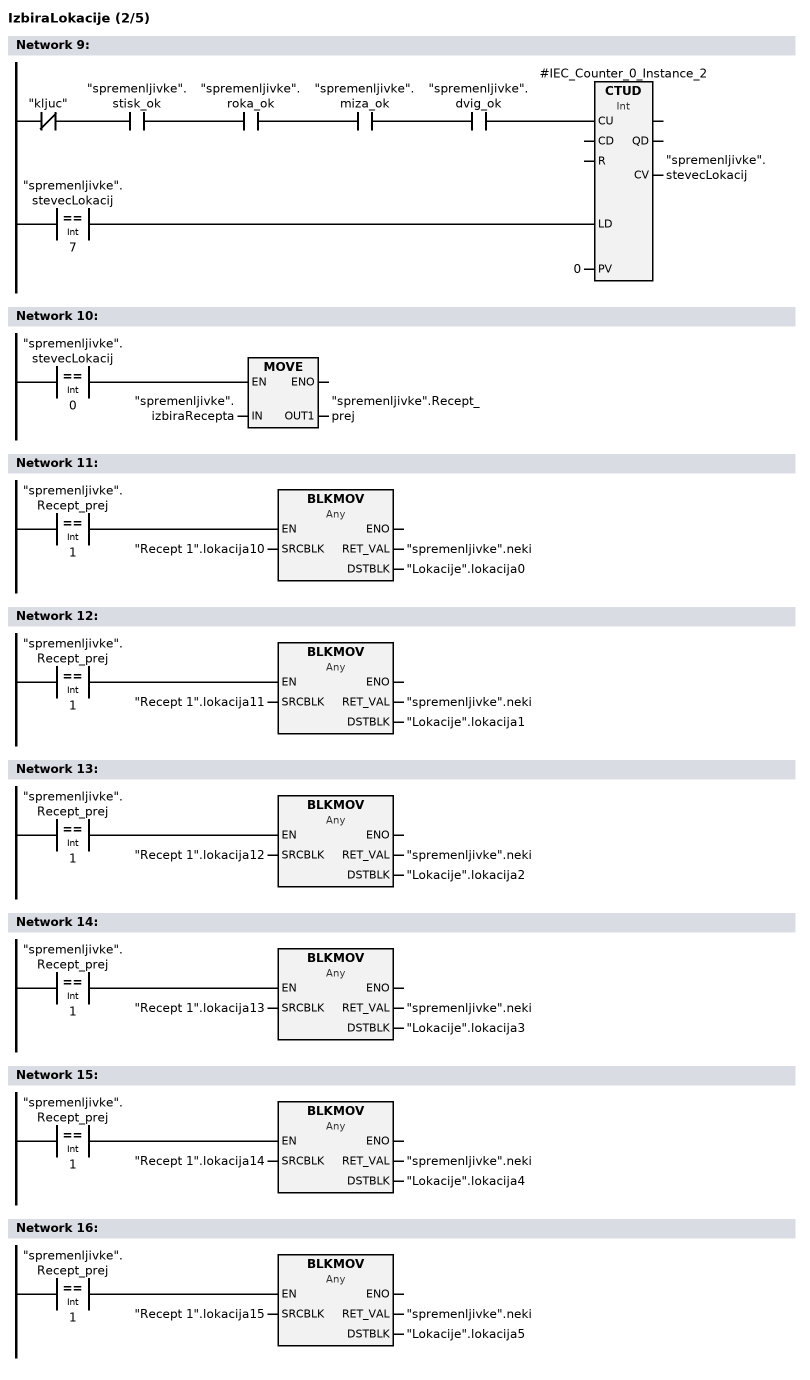
   #IEC_Counter_0_Instance_2.CTUD(CU := NOT "kljuc" AND "spremenljivke".stisk_ok AND "spremenljivke".roka_ok AND "spremenljivke".miza_ok AND "spremenljivke".dvig_ok,
                           LD := "spremenljivke".stevecLokacij = 7,
                           PV := 0,
                           CV => "spremenljivke".stevecLokacij);
END_REGION

REGION Network 10
   RUNG wire#powerrail
      { S7_Templates := "SrcType := Int" } EQ_Contact(in1 := "spremenljivke".stevecLokacij, in2 := 0)
      { S7_GenerateENO := "TRUE" } Move(in := "spremenljivke".izbiraRecepta, out1 => "spremenljivke".Recept_prej)
   END_RUNG
   // the same network as SCL:
   IF "spremenljivke".stevecLokacij = 0 THEN
       "spremenljivke".Recept_prej := "spremenljivke".izbiraRecepta;
   END_IF;
END_REGION

REGION Network 11
   IF "spremenljivke".Recept_prej = 1 THEN
       "spremenljivke".neki := BLKMOV(SRCBLK := "Recept 1".lokacija10, DSTBLK => "Lokacije".lokacija0);
   END_IF;
END_REGION

REGION Network 12
   IF "spremenljivke".Recept_prej = 1 THEN
       "spremenljivke".neki := BLKMOV(SRCBLK := "Recept 1".lokacija11, DSTBLK => "Lokacije".lokacija1);
   END_IF;
END_REGION

REGION Network 13
   IF "spremenljivke".Recept_prej = 1 THEN
       "spremenljivke".neki := BLKMOV(SRCBLK := "Recept 1".lokacija12, DSTBLK => "Lokacije".lokacija2);
   END_IF;
END_REGION

REGION Network 14
   IF "spremenljivke".Recept_prej = 1 THEN
       "spremenljivke".neki := BLKMOV(SRCBLK := "Recept 1".lokacija13, DSTBLK => "Lokacije".lokacija3);
   END_IF;
END_REGION

REGION Network 15
   IF "spremenljivke".Recept_prej = 1 THEN
       "spremenljivke".neki := BLKMOV(SRCBLK := "Recept 1".lokacija14, DSTBLK => "Lokacije".lokacija4);
   END_IF;
END_REGION

REGION Network 16
   IF "spremenljivke".Recept_prej = 1 THEN
       "spremenljivke".neki := BLKMOV(SRCBLK := "Recept 1".lokacija15, DSTBLK => "Lokacije".lokacija5);
   END_IF;
END_REGION

REGION Network 17
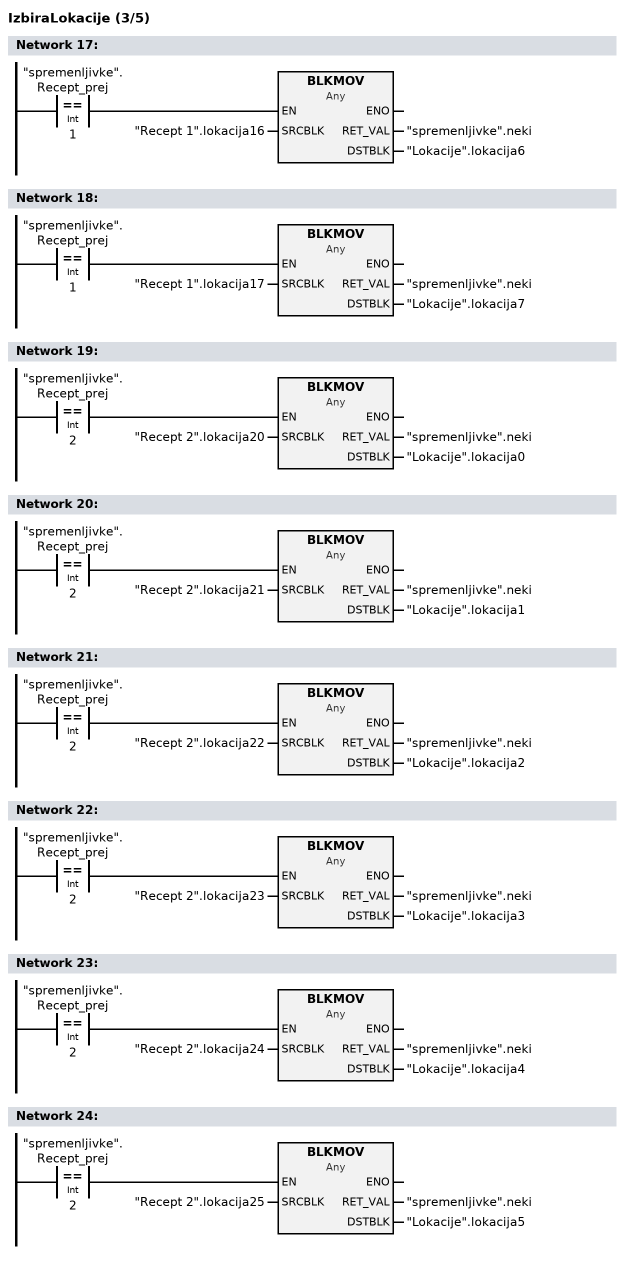
   IF "spremenljivke".Recept_prej = 1 THEN
       "spremenljivke".neki := BLKMOV(SRCBLK := "Recept 1".lokacija16, DSTBLK => "Lokacije".lokacija6);
   END_IF;
END_REGION

REGION Network 18
   IF "spremenljivke".Recept_prej = 1 THEN
       "spremenljivke".neki := BLKMOV(SRCBLK := "Recept 1".lokacija17, DSTBLK => "Lokacije".lokacija7);
   END_IF;
END_REGION

REGION Network 19
   IF "spremenljivke".Recept_prej = 2 THEN
       "spremenljivke".neki := BLKMOV(SRCBLK := "Recept 2".lokacija20, DSTBLK => "Lokacije".lokacija0);
   END_IF;
END_REGION

REGION Network 20
   IF "spremenljivke".Recept_prej = 2 THEN
       "spremenljivke".neki := BLKMOV(SRCBLK := "Recept 2".lokacija21, DSTBLK => "Lokacije".lokacija1);
   END_IF;
END_REGION

REGION Network 21
   IF "spremenljivke".Recept_prej = 2 THEN
       "spremenljivke".neki := BLKMOV(SRCBLK := "Recept 2".lokacija22, DSTBLK => "Lokacije".lokacija2);
   END_IF;
END_REGION

REGION Network 22
   IF "spremenljivke".Recept_prej = 2 THEN
       "spremenljivke".neki := BLKMOV(SRCBLK := "Recept 2".lokacija23, DSTBLK => "Lokacije".lokacija3);
   END_IF;
END_REGION

REGION Network 23
   IF "spremenljivke".Recept_prej = 2 THEN
       "spremenljivke".neki := BLKMOV(SRCBLK := "Recept 2".lokacija24, DSTBLK => "Lokacije".lokacija4);
   END_IF;
END_REGION

REGION Network 24
   IF "spremenljivke".Recept_prej = 2 THEN
       "spremenljivke".neki := BLKMOV(SRCBLK := "Recept 2".lokacija25, DSTBLK => "Lokacije".lokacija5);
   END_IF;
END_REGION

REGION Network 25
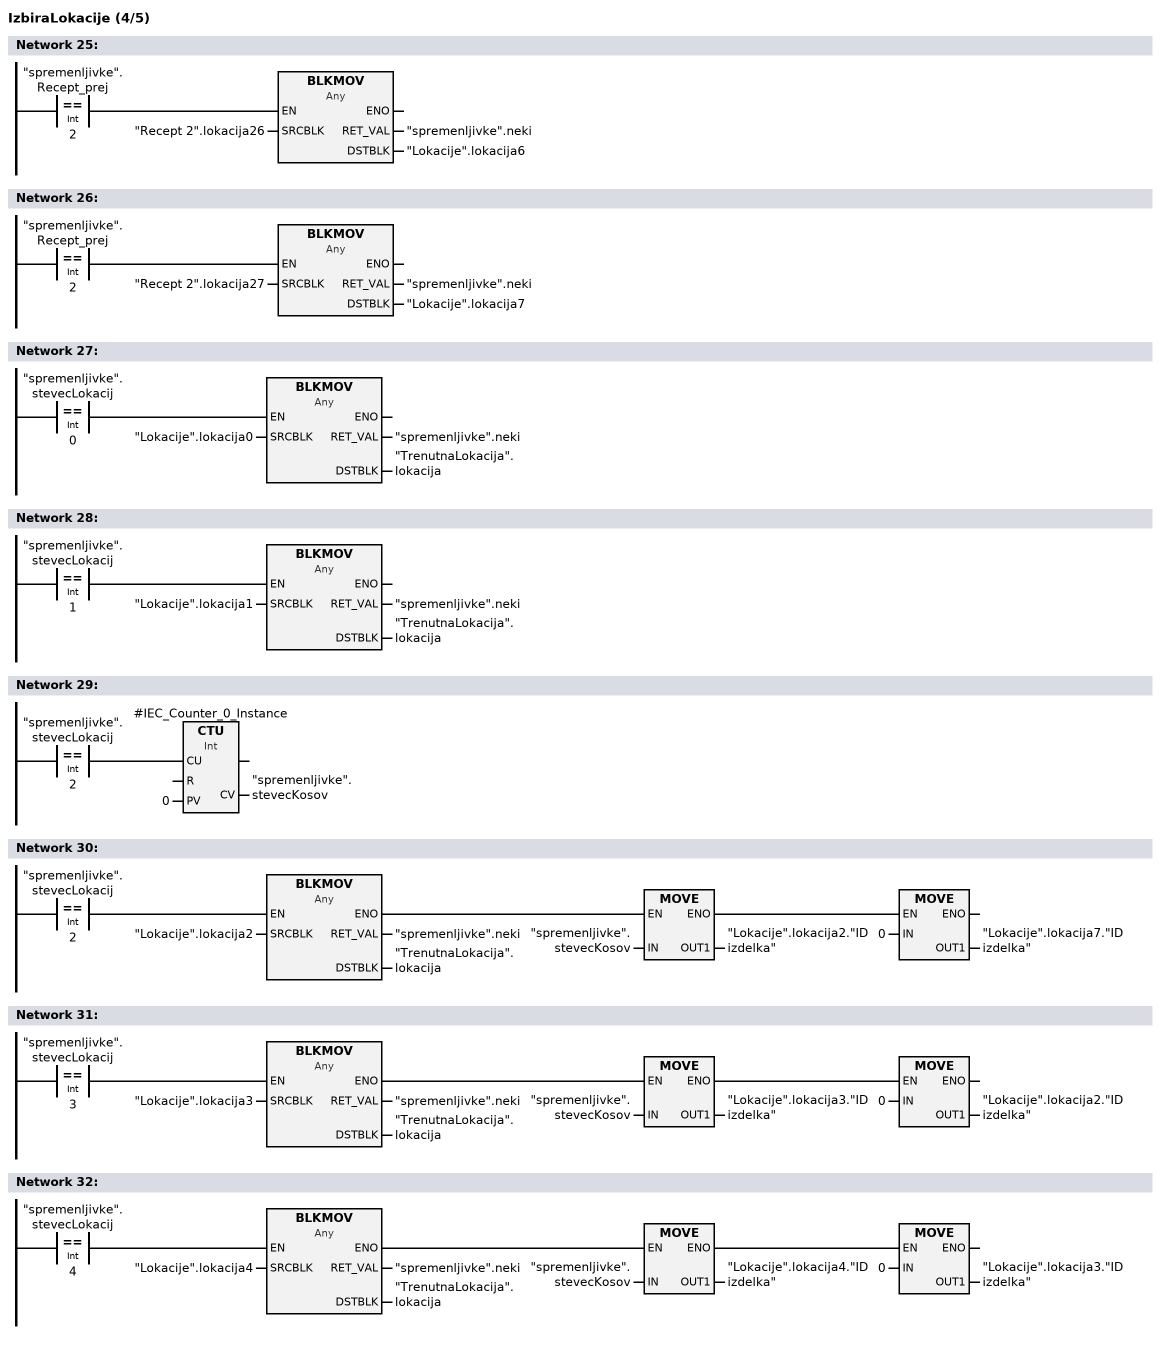
   IF "spremenljivke".Recept_prej = 2 THEN
       "spremenljivke".neki := BLKMOV(SRCBLK := "Recept 2".lokacija26, DSTBLK => "Lokacije".lokacija6);
   END_IF;
END_REGION

REGION Network 26
   IF "spremenljivke".Recept_prej = 2 THEN
       "spremenljivke".neki := BLKMOV(SRCBLK := "Recept 2".lokacija27, DSTBLK => "Lokacije".lokacija7);
   END_IF;
END_REGION

REGION Network 27
   IF "spremenljivke".stevecLokacij = 0 THEN
       "spremenljivke".neki := BLKMOV(SRCBLK := "Lokacije".lokacija0, DSTBLK => "TrenutnaLokacija".lokacija);
   END_IF;
END_REGION

REGION Network 28
   IF "spremenljivke".stevecLokacij = 1 THEN
       "spremenljivke".neki := BLKMOV(SRCBLK := "Lokacije".lokacija1, DSTBLK => "TrenutnaLokacija".lokacija);
   END_IF;
END_REGION

REGION Network 29
   #IEC_Counter_0_Instance.CTU(CU := "spremenljivke".stevecLokacij = 2,
                           PV := 0,
                           CV => "spremenljivke".stevecKosov);
END_REGION

REGION Network 30
   // ENO of a box is taken as its EN; it also drops when the box reports an error
   #_w1 := "spremenljivke".stevecLokacij = 2;
   IF #_w1 THEN
       "spremenljivke".neki := BLKMOV(SRCBLK := "Lokacije".lokacija2, DSTBLK => "TrenutnaLokacija".lokacija);
       "Lokacije".lokacija2."ID izdelka" := "spremenljivke".stevecKosov;
       "Lokacije".lokacija7."ID izdelka" := 0;
   END_IF;
END_REGION

REGION Network 31
   // ENO of a box is taken as its EN; it also drops when the box reports an error
   #_w1 := "spremenljivke".stevecLokacij = 3;
   IF #_w1 THEN
       "spremenljivke".neki := BLKMOV(SRCBLK := "Lokacije".lokacija3, DSTBLK => "TrenutnaLokacija".lokacija);
       "Lokacije".lokacija3."ID izdelka" := "spremenljivke".stevecKosov;
       "Lokacije".lokacija2."ID izdelka" := 0;
   END_IF;
END_REGION

REGION Network 32
   // ENO of a box is taken as its EN; it also drops when the box reports an error
   #_w1 := "spremenljivke".stevecLokacij = 4;
   IF #_w1 THEN
       "spremenljivke".neki := BLKMOV(SRCBLK := "Lokacije".lokacija4, DSTBLK => "TrenutnaLokacija".lokacija);
       "Lokacije".lokacija4."ID izdelka" := "spremenljivke".stevecKosov;
       "Lokacije".lokacija3."ID izdelka" := 0;
   END_IF;
END_REGION

REGION Network 33
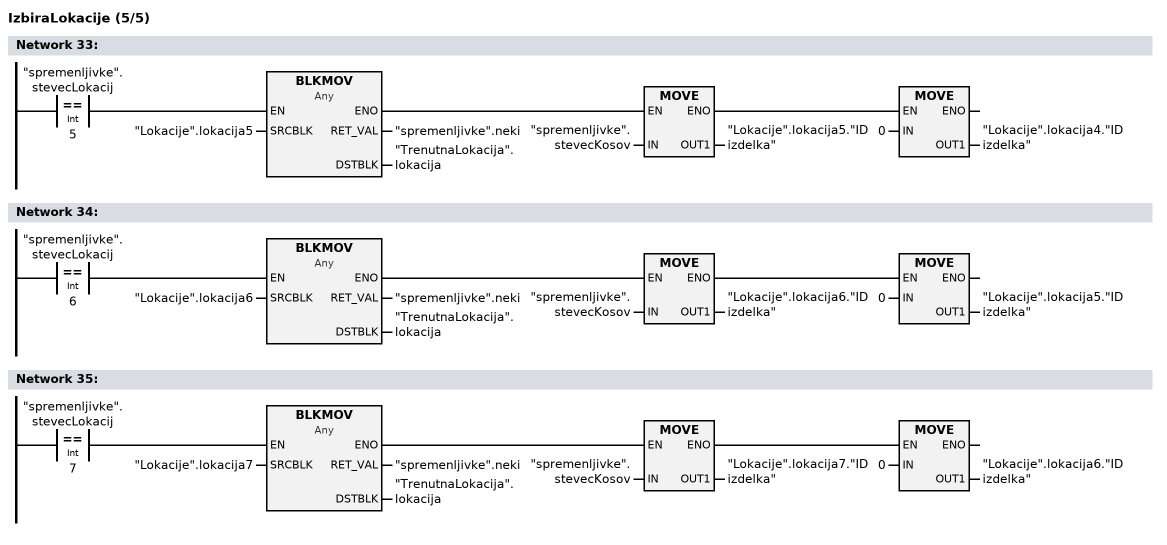
   // ENO of a box is taken as its EN; it also drops when the box reports an error
   #_w1 := "spremenljivke".stevecLokacij = 5;
   IF #_w1 THEN
       "spremenljivke".neki := BLKMOV(SRCBLK := "Lokacije".lokacija5, DSTBLK => "TrenutnaLokacija".lokacija);
       "Lokacije".lokacija5."ID izdelka" := "spremenljivke".stevecKosov;
       "Lokacije".lokacija4."ID izdelka" := 0;
   END_IF;
END_REGION

REGION Network 34
   // ENO of a box is taken as its EN; it also drops when the box reports an error
   #_w1 := "spremenljivke".stevecLokacij = 6;
   IF #_w1 THEN
       "spremenljivke".neki := BLKMOV(SRCBLK := "Lokacije".lokacija6, DSTBLK => "TrenutnaLokacija".lokacija);
       "Lokacije".lokacija6."ID izdelka" := "spremenljivke".stevecKosov;
       "Lokacije".lokacija5."ID izdelka" := 0;
   END_IF;
END_REGION

REGION Network 35
   // ENO of a box is taken as its EN; it also drops when the box reports an error
   #_w1 := "spremenljivke".stevecLokacij = 7;
   IF #_w1 THEN
       "spremenljivke".neki := BLKMOV(SRCBLK := "Lokacije".lokacija7, DSTBLK => "TrenutnaLokacija".lokacija);
       "Lokacije".lokacija7."ID izdelka" := "spremenljivke".stevecKosov;
       "Lokacije".lokacija6."ID izdelka" := 0;
   END_IF;
END_REGION
END_FUNCTION_BLOCK

FUNCTION_BLOCK "izbiraAlarmov"   // FB8, LAD
{ S7_Optimized_Access := 'FALSE' }
VERSION : 0.1
BEGIN

REGION Network 1
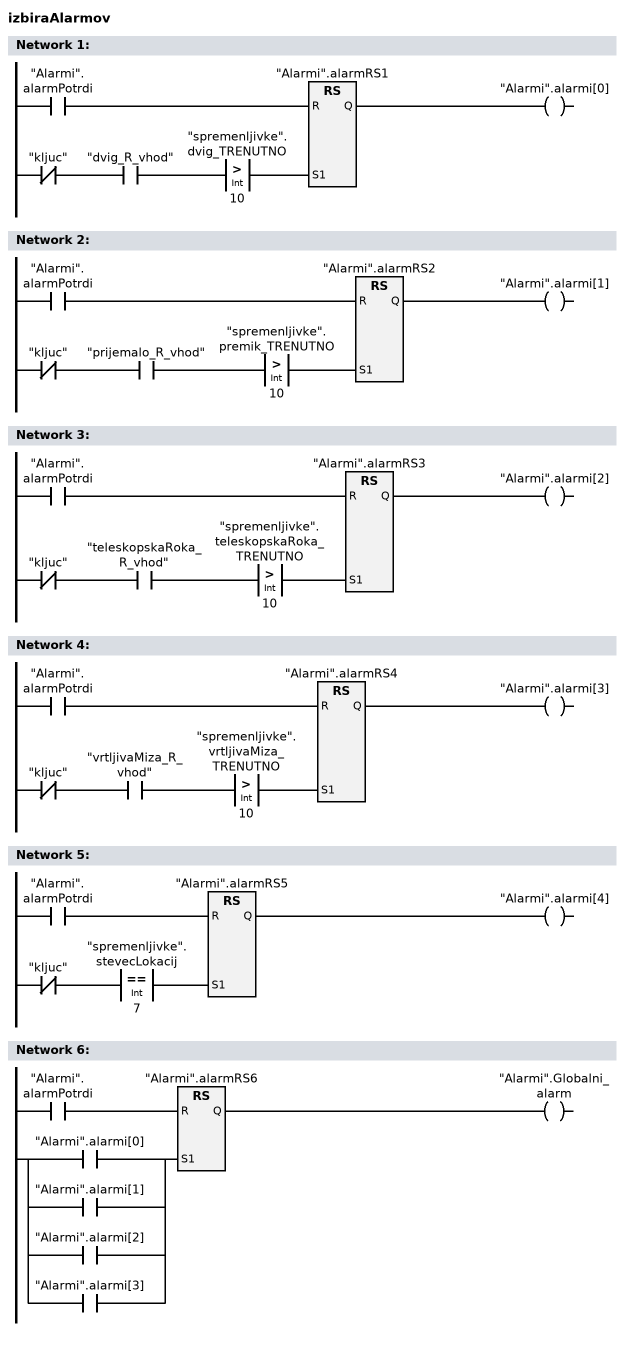
   RUNG wire#powerrail
      Contact( "Alarmi".alarmPotrdi )
      S_RS(operand := "Alarmi".alarmRS1, s1 := wire#w1)
      Coil( "Alarmi".alarmi[0] )
   END_RUNG
   RUNG wire#powerrail
      I_Contact( "kljuc" )
      Contact( "dvig_R_vhod" )
      { S7_Templates := "SrcType := Int" } GT_Contact(in1 := "spremenljivke".dvig_TRENUTNO, in2 := 10)
   END_RUNG wire#w1
   // the same network as SCL:
   IF "Alarmi".alarmPotrdi THEN
       "Alarmi".alarmRS1 := FALSE;   // RS flip-flop
   END_IF;
   IF NOT "kljuc" AND "dvig_R_vhod" AND ("spremenljivke".dvig_TRENUTNO > 10) THEN
       "Alarmi".alarmRS1 := TRUE;
   END_IF;
   "Alarmi".alarmi[0] := "Alarmi".alarmRS1;
END_REGION

REGION Network 2
   RUNG wire#powerrail
      Contact( "Alarmi".alarmPotrdi )
      S_RS(operand := "Alarmi".alarmRS2, s1 := wire#w1)
      Coil( "Alarmi".alarmi[1] )
   END_RUNG
   RUNG wire#powerrail
      I_Contact( "kljuc" )
      Contact( "prijemalo_R_vhod" )
      { S7_Templates := "SrcType := Int" } GT_Contact(in1 := "spremenljivke".premik_TRENUTNO, in2 := 10)
   END_RUNG wire#w1
   // the same network as SCL:
   IF "Alarmi".alarmPotrdi THEN
       "Alarmi".alarmRS2 := FALSE;   // RS flip-flop
   END_IF;
   IF NOT "kljuc" AND "prijemalo_R_vhod" AND ("spremenljivke".premik_TRENUTNO > 10) THEN
       "Alarmi".alarmRS2 := TRUE;
   END_IF;
   "Alarmi".alarmi[1] := "Alarmi".alarmRS2;
END_REGION

REGION Network 3
   RUNG wire#powerrail
      Contact( "Alarmi".alarmPotrdi )
      S_RS(operand := "Alarmi".alarmRS3, s1 := wire#w1)
      Coil( "Alarmi".alarmi[2] )
   END_RUNG
   RUNG wire#powerrail
      I_Contact( "kljuc" )
      Contact( "teleskopskaRoka_R_vhod" )
      { S7_Templates := "SrcType := Int" } GT_Contact(in1 := "spremenljivke".teleskopskaRoka_TRENUTNO, in2 := 10)
   END_RUNG wire#w1
   // the same network as SCL:
   IF "Alarmi".alarmPotrdi THEN
       "Alarmi".alarmRS3 := FALSE;   // RS flip-flop
   END_IF;
   IF NOT "kljuc" AND "teleskopskaRoka_R_vhod" AND ("spremenljivke".teleskopskaRoka_TRENUTNO > 10) THEN
       "Alarmi".alarmRS3 := TRUE;
   END_IF;
   "Alarmi".alarmi[2] := "Alarmi".alarmRS3;
END_REGION

REGION Network 4
   RUNG wire#powerrail
      Contact( "Alarmi".alarmPotrdi )
      S_RS(operand := "Alarmi".alarmRS4, s1 := wire#w1)
      Coil( "Alarmi".alarmi[3] )
   END_RUNG
   RUNG wire#powerrail
      I_Contact( "kljuc" )
      Contact( "vrtljivaMiza_R_vhod" )
      { S7_Templates := "SrcType := Int" } GT_Contact(in1 := "spremenljivke".vrtljivaMiza_TRENUTNO, in2 := 10)
   END_RUNG wire#w1
   // the same network as SCL:
   IF "Alarmi".alarmPotrdi THEN
       "Alarmi".alarmRS4 := FALSE;   // RS flip-flop
   END_IF;
   IF NOT "kljuc" AND "vrtljivaMiza_R_vhod" AND ("spremenljivke".vrtljivaMiza_TRENUTNO > 10) THEN
       "Alarmi".alarmRS4 := TRUE;
   END_IF;
   "Alarmi".alarmi[3] := "Alarmi".alarmRS4;
END_REGION

REGION Network 5
   RUNG wire#powerrail
      Contact( "Alarmi".alarmPotrdi )
      S_RS(operand := "Alarmi".alarmRS5, s1 := wire#w1)
      Coil( "Alarmi".alarmi[4] )
   END_RUNG
   RUNG wire#powerrail
      I_Contact( "kljuc" )
      { S7_Templates := "SrcType := Int" } EQ_Contact(in1 := "spremenljivke".stevecLokacij, in2 := 7)
   END_RUNG wire#w1
   // the same network as SCL:
   IF "Alarmi".alarmPotrdi THEN
       "Alarmi".alarmRS5 := FALSE;   // RS flip-flop
   END_IF;
   IF NOT "kljuc" AND ("spremenljivke".stevecLokacij = 7) THEN "Alarmi".alarmRS5 := TRUE; END_IF;
   "Alarmi".alarmi[4] := "Alarmi".alarmRS5;
END_REGION

REGION Network 6
   RUNG wire#powerrail
      Contact( "Alarmi".alarmPotrdi )
      S_RS(operand := "Alarmi".alarmRS6, s1 := wire#w1)
      Coil( "Alarmi".Globalni_alarm )
   END_RUNG
   RUNG wire#powerrail
      Contact( "Alarmi".alarmi[0] )
   END_RUNG wire#w1
   RUNG wire#powerrail
      Contact( "Alarmi".alarmi[1] )
   END_RUNG wire#w1
   RUNG wire#powerrail
      Contact( "Alarmi".alarmi[2] )
   END_RUNG wire#w1
   RUNG wire#powerrail
      Contact( "Alarmi".alarmi[3] )
   END_RUNG wire#w1
   // the same network as SCL:
   IF "Alarmi".alarmPotrdi THEN
       "Alarmi".alarmRS6 := FALSE;   // RS flip-flop
   END_IF;
   IF "Alarmi".alarmi[0] OR "Alarmi".alarmi[1] OR "Alarmi".alarmi[2] OR "Alarmi".alarmi[3] THEN
       "Alarmi".alarmRS6 := TRUE;
   END_IF;
   "Alarmi".Globalni_alarm := "Alarmi".alarmRS6;
END_REGION
END_FUNCTION_BLOCK

ORGANIZATION_BLOCK "Main"   // OB1, LAD
TITLE = "Main Program Sweep (Cycle)"
{ S7_Optimized_Access := 'FALSE' }
VERSION : 0.1
BEGIN

REGION Network 1
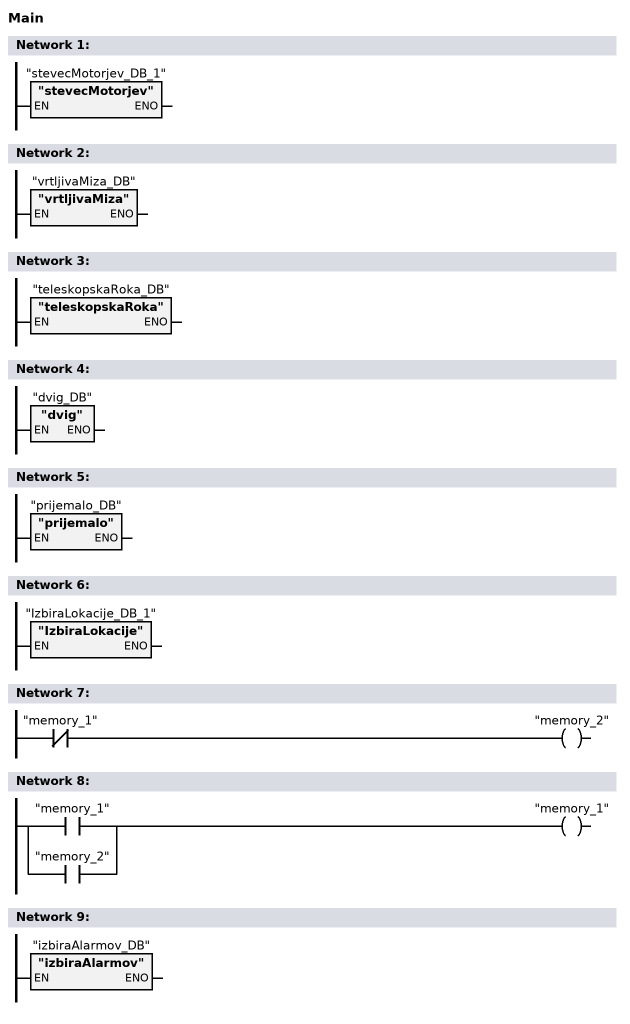
   RUNG wire#powerrail
      "stevecMotorjev_DB_1"()
   END_RUNG
   // the same network as SCL:
   "stevecMotorjev_DB_1"();   // "stevecMotorjev"
END_REGION

REGION Network 2
   RUNG wire#powerrail
      "vrtljivaMiza_DB"()
   END_RUNG
   // the same network as SCL:
   "vrtljivaMiza_DB"();   // "vrtljivaMiza"
END_REGION

REGION Network 3
   RUNG wire#powerrail
      "teleskopskaRoka_DB"()
   END_RUNG
   // the same network as SCL:
   "teleskopskaRoka_DB"();   // "teleskopskaRoka"
END_REGION

REGION Network 4
   RUNG wire#powerrail
      "dvig_DB"()
   END_RUNG
   // the same network as SCL:
   "dvig_DB"();   // "dvig"
END_REGION

REGION Network 5
   RUNG wire#powerrail
      "prijemalo_DB"()
   END_RUNG
   // the same network as SCL:
   "prijemalo_DB"();   // "prijemalo"
END_REGION

REGION Network 6
   RUNG wire#powerrail
      "IzbiraLokacije_DB_1"()
   END_RUNG
   // the same network as SCL:
   "IzbiraLokacije_DB_1"();   // "IzbiraLokacije"
END_REGION

REGION Network 7
   RUNG wire#powerrail
      I_Contact( "memory_1" )
      Coil( "memory_2" )
   END_RUNG
   // the same network as SCL:
   "memory_2" := NOT "memory_1";
END_REGION

REGION Network 8
   RUNG wire#powerrail
      Contact( "memory_1" )
      wire#w1
      Coil( "memory_1" )
   END_RUNG
   RUNG wire#powerrail
      Contact( "memory_2" )
   END_RUNG wire#w1
   // the same network as SCL:
   "memory_1" := "memory_1" OR "memory_2";
END_REGION

REGION Network 9
   RUNG wire#powerrail
      "izbiraAlarmov_DB"()
   END_RUNG
   // the same network as SCL:
   "izbiraAlarmov_DB"();   // "izbiraAlarmov"
END_REGION
END_ORGANIZATION_BLOCK

(* ===== HMI "HMI_RT_1" =====
connection "HMI_Connection_1": ETHERNET, SIMATIC S7 300/400 MPI

HMI tags "Default tag table"
   "dvig_Trenutno" : Int, 100 ms
   "kljuc" : Bool = PLC "kljuc", 100 ms
   "spremenljivke_dvig_max" : Int, 100 ms
   "spremenljivke_vrtljivaMiza_max" : Int, 100 ms
   "spremenljivke_vrtljivaMiza_TRENUTNO" : Int, 100 ms
   "spremenljivke_premik_max" : Int, 100 ms
   "spremenljivke_premik_TRENUTNO" : Int, 100 ms
   "spremenljivke_teleskopskaRoka_MAX" : Int, 100 ms
   "spremenljivke_teleskopskaRoka_TRENUTNO" : Int, 100 ms
   "vrtljivaMiza_I_vhod" : Bool = PLC "vrtljivaMiza_I_vhod", 100 ms
   "vrtljivaMiza_R_vhod" : Bool = PLC "vrtljivaMiza_R_vhod", 100 ms
   "prijemalo_I_vhod" : Bool = PLC "prijemalo_I_vhod", 100 ms
   "dvig_R_vhod" : Bool = PLC "dvig_R_vhod", 100 ms
   "teleskopskaRoka_I_vhod" : Bool = PLC "teleskopskaRoka_I_vhod", 100 ms
   "teleskopskaRoka_R_vhod" : Bool = PLC "teleskopskaRoka_R_vhod", 100 ms
   "prijemalo_R_vhod" : Bool = PLC "prijemalo_R_vhod", 100 ms
   "dvig_I_vhod" : Bool = PLC "dvig_I_vhod", 100 ms
   "vrtljivaMiza_P_izhod" : Bool = PLC "vrtljivaMiza_P_izhod", 100 ms
   "teleskopskaRoka_P_izhod" : Bool = PLC "teleskopskaRoka_P_izhod", 100 ms
   "dvig_P_izhod" : Bool = PLC "dvig_P_izhod", 100 ms
   "prijemalo_P_izhod" : Bool = PLC "prijemalo_P_izhod", 100 ms
   "Alarmi" : Word, 100 ms
   "Alarmi_alarmRS3" : Bool, 100 ms
   "Alarmi_alarmi{3}" : Bool, 100 ms
   "Alarmi_alarmi{1}" : Bool, 100 ms
   "Alarmi_alarmi{2}" : Bool, 100 ms
   "Alarmi_alarmi{0}" : Bool, 100 ms
   "Alarmi_alarmPotrdi" : Bool, 100 ms
   "spremenljivke_izbiraRecepta" : Int, 100 ms
   "Recept 1_lokacija11_koordinate_miza" : Int, 100 ms
   "Recept 1_lokacija12_koordinate_miza" : Int, 100 ms
   "Recept 1_lokacija11_koordinate_izteg" : Int, 100 ms
   "Recept 1_lokacija12_koordinate_izteg" : Int, 100 ms
   "Recept 1_lokacija12_koordinate_dvig" : Int, 100 ms
   "Recept 2_lokacija21_koordinate_miza" : Int, 100 ms
   "Recept 2_lokacija22_koordinate_miza" : Int, 100 ms
   "Recept 2_lokacija21_koordinate_izteg" : Int, 100 ms
   "Recept 2_lokacija22_koordinate_izteg" : Int, 100 ms
   "Recept 2_lokacija22_koordinate_dvig" : Int, 100 ms
   "Recept 1_lokacija14_koordinate_miza" : Int, 100 ms
   "Recept 1_lokacija15_koordinate_miza" : Int, 100 ms
   "Recept 1_lokacija16_koordinate_miza" : Int, 100 ms
   "Recept 1_lokacija17_koordinate_miza" : Int, 100 ms
   "Recept 1_lokacija14_koordinate_izteg" : Int, 100 ms
   "Recept 1_lokacija15_koordinate_izteg" : Int, 100 ms
   "Recept 1_lokacija16_koordinate_izteg" : Int, 100 ms
   "Recept 1_lokacija17_koordinate_izteg" : Int, 100 ms
   "Recept 1_lokacija15_koordinate_dvig" : Int, 100 ms
   "Recept 1_lokacija16_koordinate_dvig" : Int, 100 ms
   "Recept 2_lokacija24_koordinate_miza" : Int, 100 ms
   "Recept 2_lokacija25_koordinate_miza" : Int, 100 ms
   "Recept 2_lokacija26_koordinate_miza" : Int, 100 ms
   "Recept 2_lokacija27_koordinate_miza" : Int, 100 ms
   "Recept 2_lokacija24_koordinate_izteg" : Int, 100 ms
   "Recept 2_lokacija25_koordinate_izteg" : Int, 100 ms
   "Recept 2_lokacija26_koordinate_izteg" : Int, 100 ms
   "Recept 2_lokacija27_koordinate_izteg" : Int, 100 ms
   "Recept 2_lokacija25_koordinate_dvig" : Int, 100 ms
   "Recept 2_lokacija26_koordinate_dvig" : Int, 100 ms
   "Alarmi_Globalni_alarm" : Bool, 100 ms
   "spremenljivke_stevecLokacij" : Int, 1 s
   "spremenljivke_stevecKosov" : Int, 1 s

discrete alarms
   1: '', class Errors, trigger "Alarmi" bit 8
   2: '', class Errors, trigger "Alarmi" bit 9
   3: '', class Errors, trigger "Alarmi" bit 10
   4: '', class Errors, trigger "Alarmi" bit 11
   5: '', class Warnings, trigger "Alarmi" bit 12

screen "Pregled" 1440x900, template "Template_1"
   GraphicView "Graphic view_1" at 302,51 size 899x707
   Switch "Switch_1" at 663,678 size 105x63
   Slider "Slider_4" at 866,109 size 43x121
   Slider "Slider_1" at 634,313 size 39x123
   Slider "Slider_2" at 996,91 size 43x120
   Slider "Slider_3" at 889,490 size 43x140
   GraphicView "Graphic view_2" at 921,102 size 46x36
   GraphicView "Graphic view_3" at 1059,175 size 47x37
   GraphicView "Graphic view_4" at 582,403 size 45x36
   GraphicView "Graphic view_5" at 946,567 size 47x38
   GraphicView "Graphic view_10" at 1055,117 size 51x51
   GraphicView "Graphic view_11" at 916,42 size 51x51
   GraphicView "Graphic view_12" at 583,343 size 51x51
   GraphicView "Graphic view_13" at 943,509 size 51x51
   IOField "I/O field_1" at 313,118 size 100x40
   IOField "I/O field_7" at 218,227 size 76x30
   IOField "I/O field_8" at 223,255 size 67x34
   IOField "I/O field_9" at 220,202 size 74x25
   IOField "I/O field_12" at 223,322 size 65x30
   IOField "I/O field_11" at 223,372 size 63x36
   IOField "I/O field_10" at 226,345 size 55x38
   IOField "I/O field_2" at 218,202 size 74x25
   IOField "I/O field_3" at 216,225 size 76x30
   IOField "I/O field_4" at 223,255 size 67x34
   IOField "I/O field_5" at 226,345 size 55x38
   IOField "I/O field_6" at 221,322 size 65x30
   IOField "I/O field_13" at 223,372 size 63x32
   IOField "I/O field_14" at 389,423 size 100x40
   IOField "I/O field_15" at 474,467 size 66x44
   TextField "Text field_12" at 780,698 size 639x37
   TextField "Text field_13" at 245,693 size 145x47
   TextField "Text field_2" at 11,167 size 209x29
   TextField "Text field_1" at 4,120 size 288x34
   TextField "Text field_3" at 37,203 size 50x25
   TextField "Text field_4" at 37,230 size 117x25
   TextField "Text field_5" at 38,257 size 159x25
   TextField "Text field_6" at 11,293 size 213x29
   TextField "Text field_7" at 40,325 size 50x25
   TextField "Text field_9" at 38,376 size 159x25
   TextField "Text field_8" at 40,352 size 117x25
   TextField "Text field_10" at 0,426 size 356x34
   TextField "Text field_11" at 0,470 size 435x34

screen "Alarmi" 1440x900, template "Template_1"
   AlarmView "Alarm view_1" at 87,84 size 1250x460
   Button "Button_1" at 554,634 size 309x73

screen "Recepti" 1440x900, template "Template_1"
   Button "Button_1" at 156,72 size 290x90
   Button "Button_2" at 690,88 size 138x50
   Button "Button_3" at 980,88 size 138x50
   Button "Button_4" at 37,391 size 404x86
   Button "Button_5" at 8,550 size 450x112
   Button "Button_6" at 503,236 size 242x60
   Button "Button_7" at 789,236 size 276x60
   Button "Button_8" at 1076,236 size 242x60
   IOField "I/O field_1" at 511,400 size 238x62
   IOField "I/O field_2" at 520,580 size 238x62
   IOField "I/O field_3" at 797,400 size 238x62
   IOField "I/O field_4" at 803,580 size 238x62
   IOField "I/O field_5" at 1091,400 size 238x62
   IOField "I/O field_6" at 1096,580 size 238x62
   IOField "I/O field_7" at 511,400 size 238x62
   IOField "I/O field_8" at 797,400 size 238x62
   IOField "I/O field_9" at 1091,400 size 238x62
   IOField "I/O field_10" at 520,580 size 238x62
   IOField "I/O field_11" at 803,580 size 238x62
   IOField "I/O field_12" at 1096,580 size 238x62

Template "Template_1" 1440x900
   Button "Template_Button_1" at 190,773 size 238x62
   Button "Template_Button_2" at 590,772 size 238x62
   Button "Template_Button_3" at 981,771 size 238x62
*)